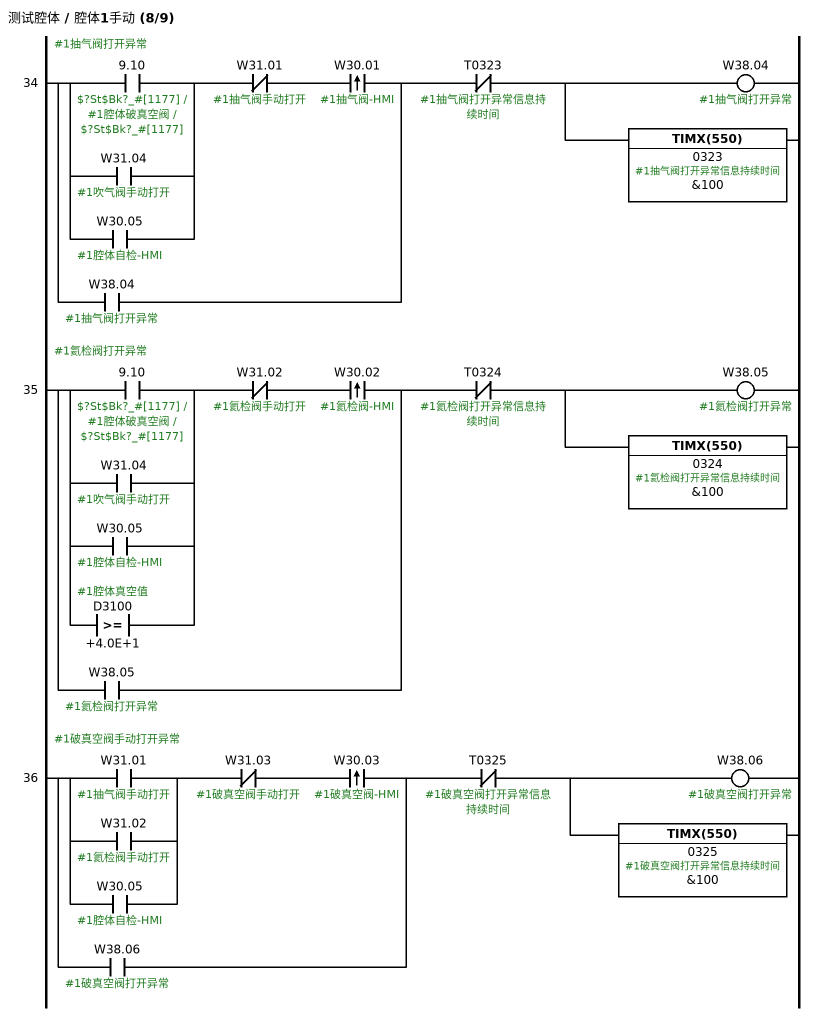
; [picture p120: 测试腔体 / 腔体1手动, rungs 34-36]
; rung 34: #1抽气阀打开异常
LD 9.10  ; $?St$Bk?_#[1177] / #1腔体破真空阀 / $?St$Bk?_#[1177]
OR W31.04  ; #1吹气阀手动打开
OR W30.05  ; #1腔体自检-HMI
ANDNOT W31.01  ; #1抽气阀手动打开
@AND W30.01  ; #1抽气阀-HMI
OR W38.04  ; #1抽气阀打开异常
ANDNOT T0323  ; #1抽气阀打开异常信息持续时间
OUT W38.04  ; #1抽气阀打开异常
TIMX(550) 0323 &100  ; #1抽气阀打开异常信息持续时间
; rung 35: #1氦检阀打开异常
LD 9.10  ; $?St$Bk?_#[1177] / #1腔体破真空阀 / $?St$Bk?_#[1177]
OR W31.04  ; #1吹气阀手动打开
OR W30.05  ; #1腔体自检-HMI
OR>=F(334) D3100 +4.0E+1  ; #1腔体真空值
ANDNOT W31.02  ; #1氦检阀手动打开
@AND W30.02  ; #1氦检阀-HMI
OR W38.05  ; #1氦检阀打开异常
ANDNOT T0324  ; #1氦检阀打开异常信息持续时间
OUT W38.05  ; #1氦检阀打开异常
TIMX(550) 0324 &100  ; #1氦检阀打开异常信息持续时间
; rung 36: #1破真空阀手动打开异常
LD W31.01  ; #1抽气阀手动打开
OR W31.02  ; #1氦检阀手动打开
OR W30.05  ; #1腔体自检-HMI
ANDNOT W31.03  ; #1破真空阀手动打开
@AND W30.03  ; #1破真空阀-HMI
OR W38.06  ; #1破真空阀打开异常
ANDNOT T0325  ; #1破真空阀打开异常信息持续时间
OUT W38.06  ; #1破真空阀打开异常
TIMX(550) 0325 &100  ; #1破真空阀打开异常信息持续时间

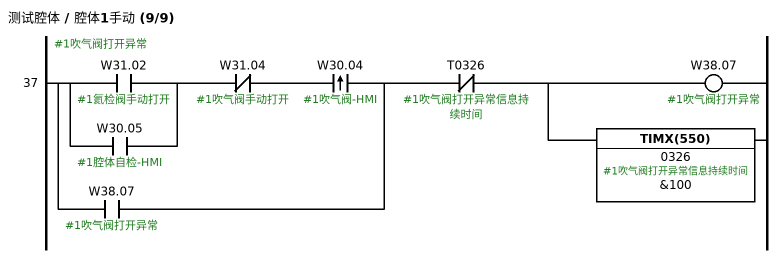
; rung 37: #1吹气阀打开异常
LD W31.02  ; #1氦检阀手动打开
OR W30.05  ; #1腔体自检-HMI
ANDNOT W31.04  ; #1吹气阀手动打开
@AND W30.04  ; #1吹气阀-HMI
OR W38.07  ; #1吹气阀打开异常
ANDNOT T0326  ; #1吹气阀打开异常信息持续时间
OUT W38.07  ; #1吹气阀打开异常
TIMX(550) 0326 &100  ; #1吹气阀打开异常信息持续时间

### Section 腔体2手动

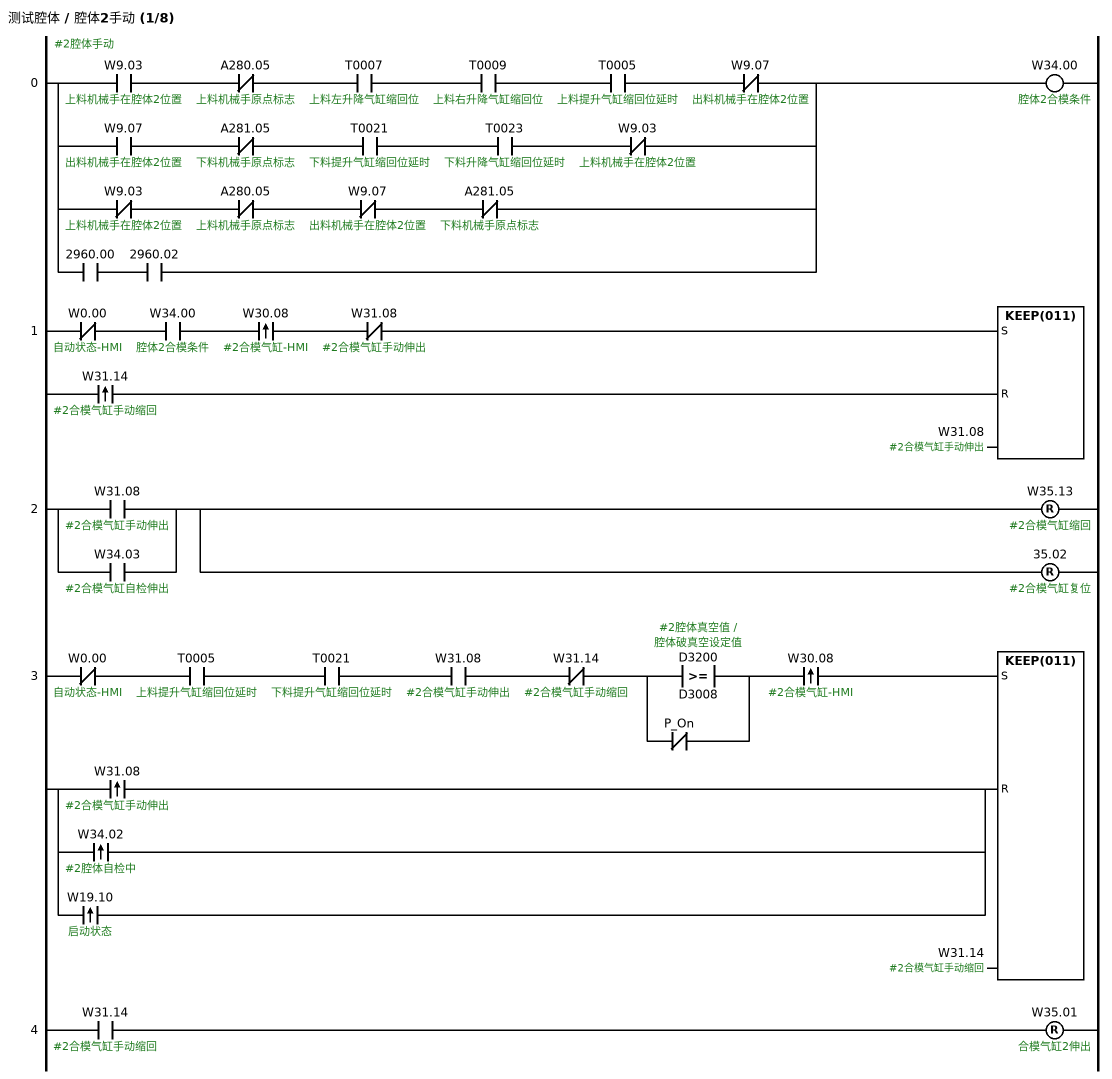
; rung 0: #2腔体手动
LD W9.03  ; 上料机械手在腔体2位置
ANDNOT A280.05  ; 上料机械手原点标志
AND T0007  ; 上料左升降气缸缩回位
AND T0009  ; 上料右升降气缸缩回位
AND T0005  ; 上料提升气缸缩回位延时
ANDNOT W9.07  ; 出料机械手在腔体2位置
LD W9.07  ; 出料机械手在腔体2位置
ANDNOT A281.05  ; 下料机械手原点标志
AND T0021  ; 下料提升气缸缩回位延时
AND T0023  ; 下料升降气缸缩回位延时
ANDNOT W9.03  ; 上料机械手在腔体2位置
ORLD
LDNOT W9.03  ; 上料机械手在腔体2位置
ANDNOT A280.05  ; 上料机械手原点标志
ANDNOT W9.07  ; 出料机械手在腔体2位置
ANDNOT A281.05  ; 下料机械手原点标志
ORLD
LD 2960.00
AND 2960.02
ORLD
OUT W34.00  ; 腔体2合模条件
; rung 1
LDNOT W0.00  ; 自动状态-HMI
AND W34.00  ; 腔体2合模条件
@AND W30.08  ; #2合模气缸-HMI
ANDNOT W31.08  ; #2合模气缸手动伸出
@LD W31.14  ; #2合模气缸手动缩回
KEEP(011) W31.08  ; #2合模气缸手动伸出
; rung 2
LD W31.08  ; #2合模气缸手动伸出
OR W34.03  ; #2合模气缸自检伸出
RSET W35.13  ; #2合模气缸缩回
RSET 35.02  ; #2合模气缸复位
; rung 3
LDNOT W0.00  ; 自动状态-HMI
AND T0005  ; 上料提升气缸缩回位延时
AND T0021  ; 下料提升气缸缩回位延时
AND W31.08  ; #2合模气缸手动伸出
ANDNOT W31.14  ; #2合模气缸手动缩回
LD>=F(334) D3200 D3008  ; #2腔体真空值, 腔体破真空设定值
ORNOT P_On
ANDLD
@AND W30.08  ; #2合模气缸-HMI
@LD W31.08  ; #2合模气缸手动伸出
@OR W34.02  ; #2腔体自检中
@OR W19.10  ; 启动状态
KEEP(011) W31.14  ; #2合模气缸手动缩回
; rung 4
LD W31.14  ; #2合模气缸手动缩回
RSET W35.01  ; 合模气缸2伸出

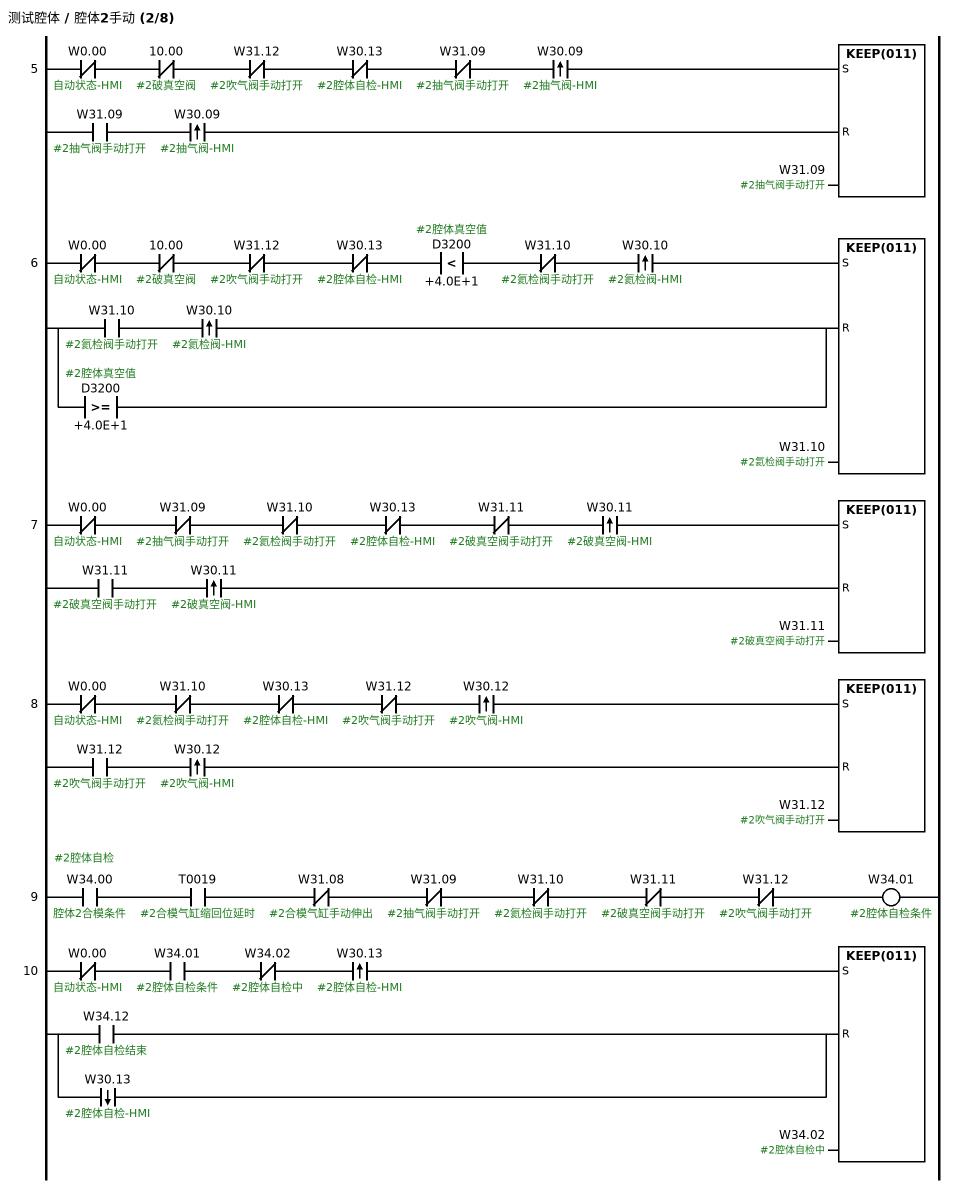
; rung 5
LDNOT W0.00  ; 自动状态-HMI
ANDNOT 10.00  ; #2破真空阀
ANDNOT W31.12  ; #2吹气阀手动打开
ANDNOT W30.13  ; #2腔体自检-HMI
ANDNOT W31.09  ; #2抽气阀手动打开
@AND W30.09  ; #2抽气阀-HMI
LD W31.09  ; #2抽气阀手动打开
@AND W30.09  ; #2抽气阀-HMI
KEEP(011) W31.09  ; #2抽气阀手动打开
; rung 6
LDNOT W0.00  ; 自动状态-HMI
ANDNOT 10.00  ; #2破真空阀
ANDNOT W31.12  ; #2吹气阀手动打开
ANDNOT W30.13  ; #2腔体自检-HMI
AND<F(331) D3200 +4.0E+1  ; #2腔体真空值
ANDNOT W31.10  ; #2氦检阀手动打开
@AND W30.10  ; #2氦检阀-HMI
LD W31.10  ; #2氦检阀手动打开
@AND W30.10  ; #2氦检阀-HMI
OR>=F(334) D3200 +4.0E+1  ; #2腔体真空值
KEEP(011) W31.10  ; #2氦检阀手动打开
; rung 7
LDNOT W0.00  ; 自动状态-HMI
ANDNOT W31.09  ; #2抽气阀手动打开
ANDNOT W31.10  ; #2氦检阀手动打开
ANDNOT W30.13  ; #2腔体自检-HMI
ANDNOT W31.11  ; #2破真空阀手动打开
@AND W30.11  ; #2破真空阀-HMI
LD W31.11  ; #2破真空阀手动打开
@AND W30.11  ; #2破真空阀-HMI
KEEP(011) W31.11  ; #2破真空阀手动打开
; rung 8
LDNOT W0.00  ; 自动状态-HMI
ANDNOT W31.10  ; #2氦检阀手动打开
ANDNOT W30.13  ; #2腔体自检-HMI
ANDNOT W31.12  ; #2吹气阀手动打开
@AND W30.12  ; #2吹气阀-HMI
LD W31.12  ; #2吹气阀手动打开
@AND W30.12  ; #2吹气阀-HMI
KEEP(011) W31.12  ; #2吹气阀手动打开
; rung 9: #2腔体自检
LD W34.00  ; 腔体2合模条件
AND T0019  ; #2合模气缸缩回位延时
ANDNOT W31.08  ; #2合模气缸手动伸出
ANDNOT W31.09  ; #2抽气阀手动打开
ANDNOT W31.10  ; #2氦检阀手动打开
ANDNOT W31.11  ; #2破真空阀手动打开
ANDNOT W31.12  ; #2吹气阀手动打开
OUT W34.01  ; #2腔体自检条件
; rung 10
LDNOT W0.00  ; 自动状态-HMI
AND W34.01  ; #2腔体自检条件
ANDNOT W34.02  ; #2腔体自检中
@AND W30.13  ; #2腔体自检-HMI
LD W34.12  ; #2腔体自检结束
%OR W30.13  ; #2腔体自检-HMI
KEEP(011) W34.02  ; #2腔体自检中

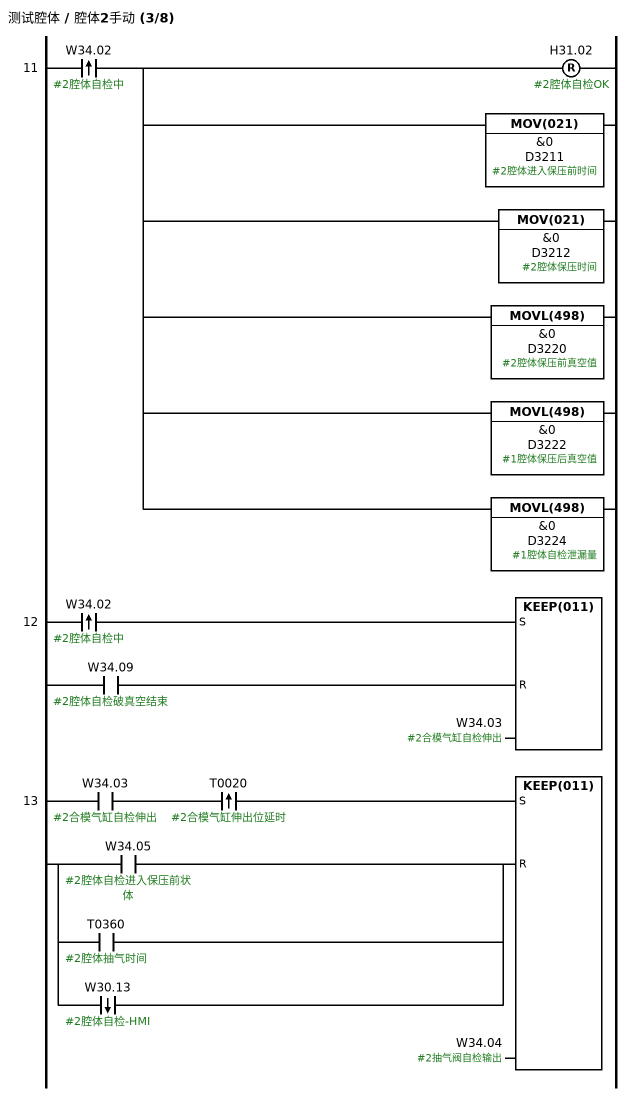
; rung 11
@LD W34.02  ; #2腔体自检中
RSET H31.02  ; #2腔体自检OK
MOV(021) &0 D3211  ; #2腔体进入保压前时间
MOV(021) &0 D3212  ; #2腔体保压时间
MOVL(498) &0 D3220  ; #2腔体保压前真空值
MOVL(498) &0 D3222  ; #1腔体保压后真空值
MOVL(498) &0 D3224  ; #1腔体自检泄漏量
; rung 12
@LD W34.02  ; #2腔体自检中
LD W34.09  ; #2腔体自检破真空结束
KEEP(011) W34.03  ; #2合模气缸自检伸出
; rung 13
LD W34.03  ; #2合模气缸自检伸出
@AND T0020  ; #2合模气缸伸出位延时
LD W34.05  ; #2腔体自检进入保压前状体
OR T0360  ; #2腔体抽气时间
%OR W30.13  ; #2腔体自检-HMI
KEEP(011) W34.04  ; #2抽气阀自检输出

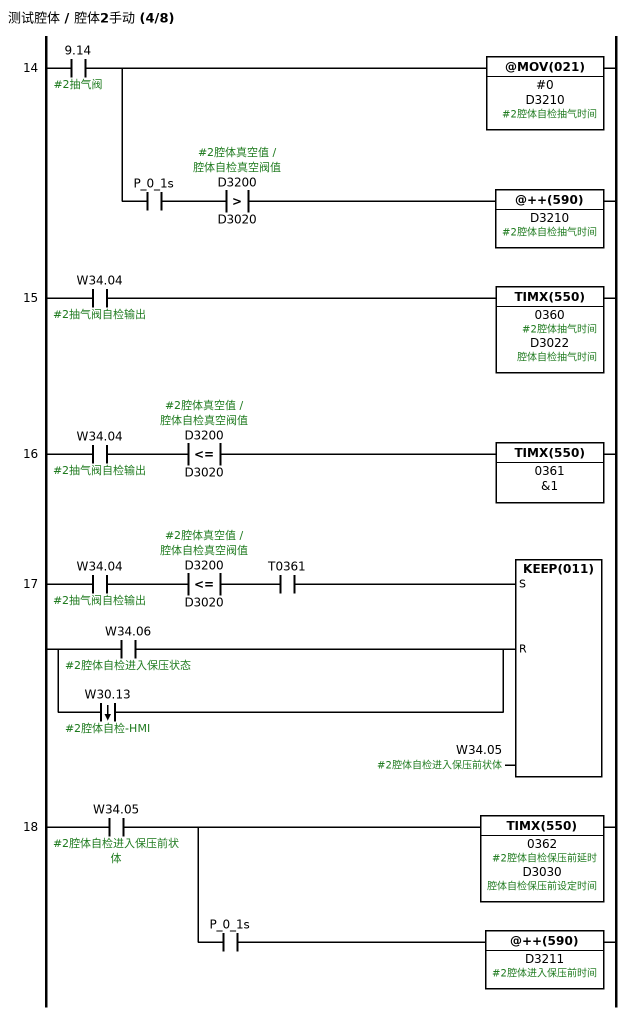
; rung 14
LD 9.14  ; #2抽气阀
@MOV(021) #0 D3210  ; #2腔体自检抽气时间
AND P_0_1s
AND>F(333) D3200 D3020  ; #2腔体真空值, 腔体自检真空阀值
@++(590) D3210  ; #2腔体自检抽气时间
; rung 15
LD W34.04  ; #2抽气阀自检输出
TIMX(550) 0360 D3022  ; 腔体自检抽气时间, #2腔体抽气时间
; rung 16
LD W34.04  ; #2抽气阀自检输出
AND<=F(332) D3200 D3020  ; #2腔体真空值, 腔体自检真空阀值
TIMX(550) 0361 &1
; rung 17
LD W34.04  ; #2抽气阀自检输出
AND<=F(332) D3200 D3020  ; #2腔体真空值, 腔体自检真空阀值
AND T0361
LD W34.06  ; #2腔体自检进入保压状态
%OR W30.13  ; #2腔体自检-HMI
KEEP(011) W34.05  ; #2腔体自检进入保压前状体
; rung 18
LD W34.05  ; #2腔体自检进入保压前状体
TIMX(550) 0362 D3030  ; 腔体自检保压前设定时间, #2腔体自检保压前延时
AND P_0_1s
@++(590) D3211  ; #2腔体进入保压前时间

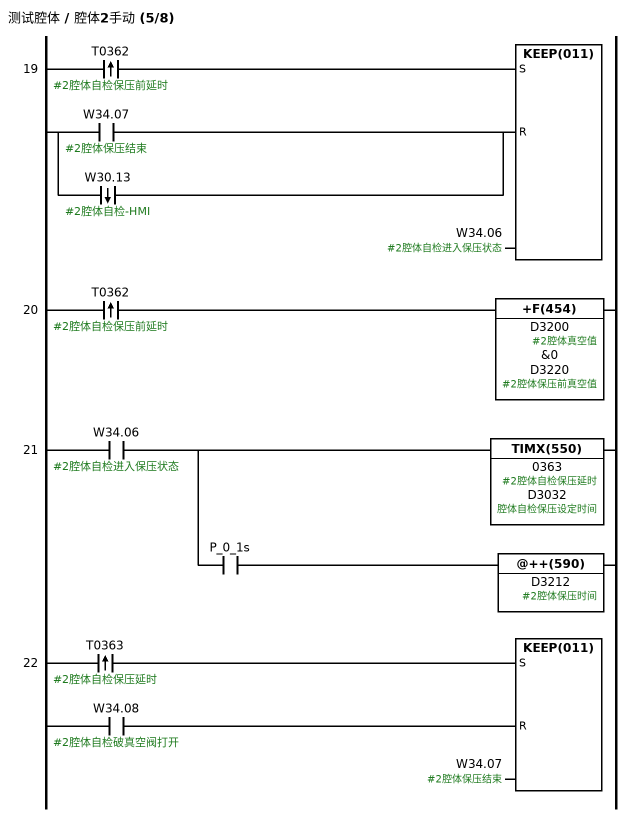
; rung 19
@LD T0362  ; #2腔体自检保压前延时
LD W34.07  ; #2腔体保压结束
%OR W30.13  ; #2腔体自检-HMI
KEEP(011) W34.06  ; #2腔体自检进入保压状态
; rung 20
@LD T0362  ; #2腔体自检保压前延时
+F(454) D3200 &0 D3220  ; #2腔体真空值, #2腔体保压前真空值
; rung 21
LD W34.06  ; #2腔体自检进入保压状态
TIMX(550) 0363 D3032  ; 腔体自检保压设定时间, #2腔体自检保压延时
AND P_0_1s
@++(590) D3212  ; #2腔体保压时间
; rung 22
@LD T0363  ; #2腔体自检保压延时
LD W34.08  ; #2腔体自检破真空阀打开
KEEP(011) W34.07  ; #2腔体保压结束

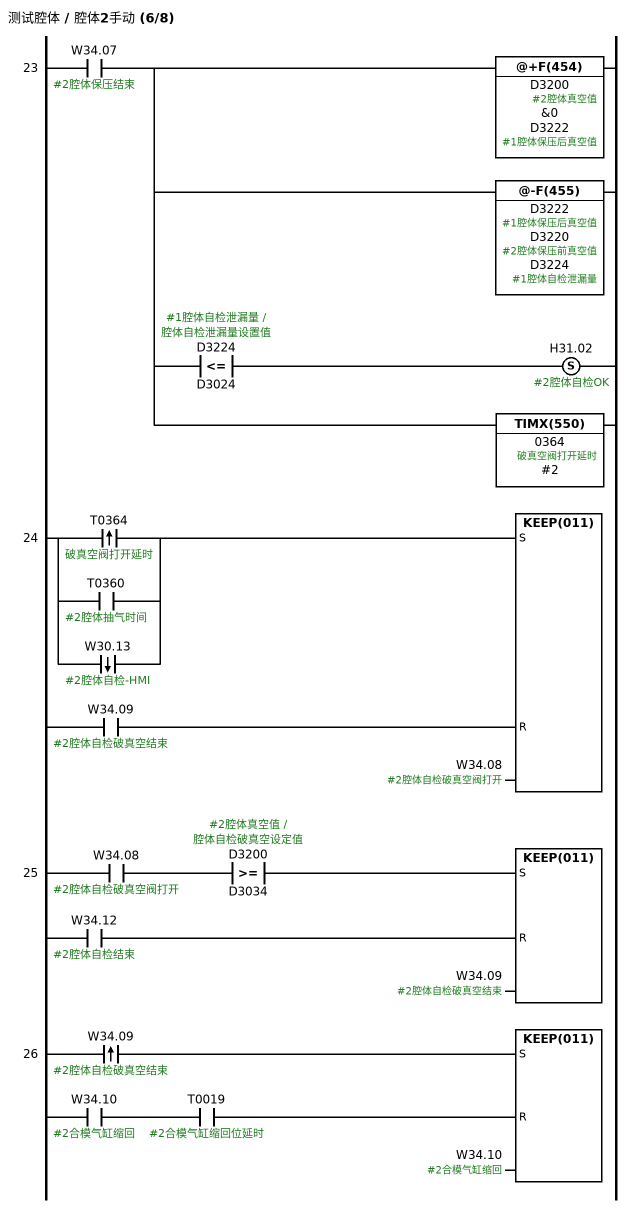
; rung 23
LD W34.07  ; #2腔体保压结束
OUT TR0
@+F(454) D3200 &0 D3222  ; #2腔体真空值, #1腔体保压后真空值
@-F(455) D3222 D3220 D3224  ; #1腔体保压后真空值, #2腔体保压前真空值, #1腔体自检泄漏量
AND<=(315) D3224 D3024  ; #1腔体自检泄漏量, 腔体自检泄漏量设置值
SET H31.02  ; #2腔体自检OK
LD TR0
TIMX(550) 0364 #2  ; 破真空阀打开延时
; rung 24
@LD T0364  ; 破真空阀打开延时
OR T0360  ; #2腔体抽气时间
%OR W30.13  ; #2腔体自检-HMI
LD W34.09  ; #2腔体自检破真空结束
KEEP(011) W34.08  ; #2腔体自检破真空阀打开
; rung 25
LD W34.08  ; #2腔体自检破真空阀打开
AND>=F(334) D3200 D3034  ; #2腔体真空值, 腔体自检破真空设定值
LD W34.12  ; #2腔体自检结束
KEEP(011) W34.09  ; #2腔体自检破真空结束
; rung 26
@LD W34.09  ; #2腔体自检破真空结束
LD W34.10  ; #2合模气缸缩回
AND T0019  ; #2合模气缸缩回位延时
KEEP(011) W34.10  ; #2合模气缸缩回

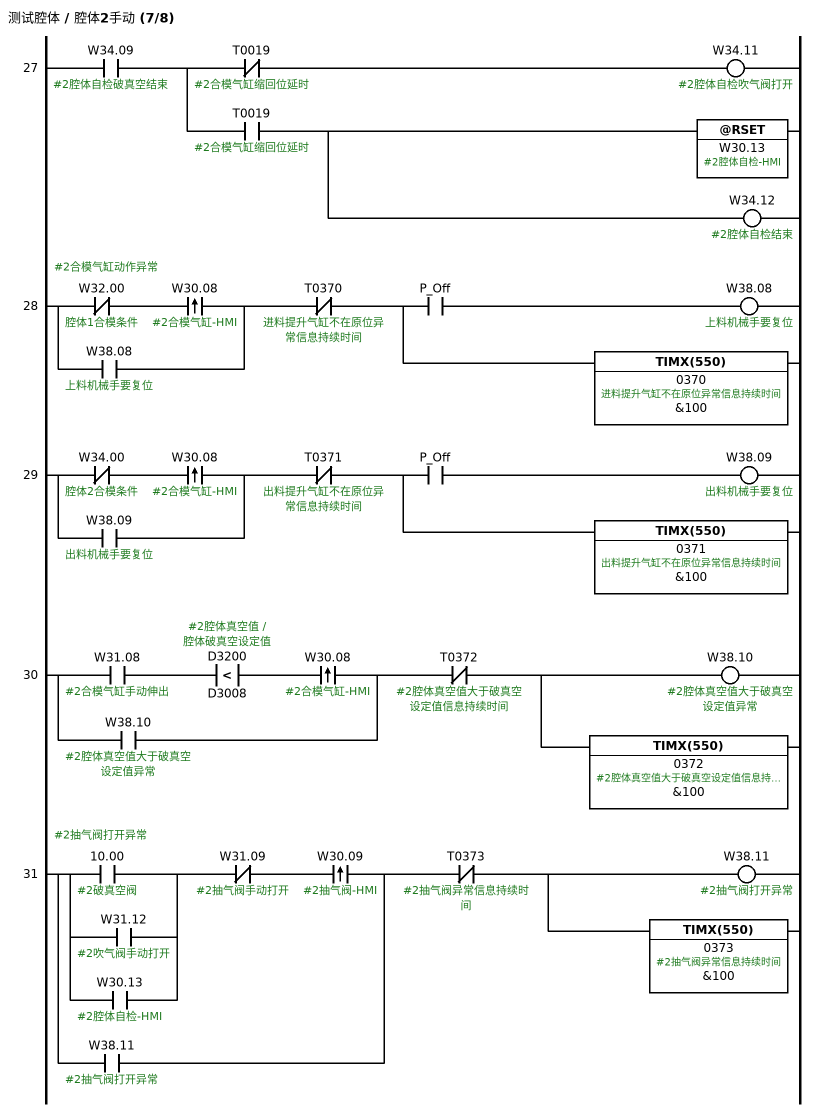
; rung 27
LD W34.09  ; #2腔体自检破真空结束
OUT TR0
ANDNOT T0019  ; #2合模气缸缩回位延时
OUT W34.11  ; #2腔体自检吹气阀打开
LD TR0
AND T0019  ; #2合模气缸缩回位延时
@RSET W30.13  ; #2腔体自检-HMI
OUT W34.12  ; #2腔体自检结束
; rung 28: #2合模气缸动作异常
LDNOT W32.00  ; 腔体1合模条件
@AND W30.08  ; #2合模气缸-HMI
OR W38.08  ; 上料机械手要复位
ANDNOT T0370  ; 进料提升气缸不在原位异常信息持续时间
OUT TR0
AND P_Off
OUT W38.08  ; 上料机械手要复位
LD TR0
TIMX(550) 0370 &100  ; 进料提升气缸不在原位异常信息持续时间
; rung 29
LDNOT W34.00  ; 腔体2合模条件
@AND W30.08  ; #2合模气缸-HMI
OR W38.09  ; 出料机械手要复位
ANDNOT T0371  ; 出料提升气缸不在原位异常信息持续时间
OUT TR0
AND P_Off
OUT W38.09  ; 出料机械手要复位
LD TR0
TIMX(550) 0371 &100  ; 出料提升气缸不在原位异常信息持续时间
; rung 30
LD W31.08  ; #2合模气缸手动伸出
AND<F(331) D3200 D3008  ; #2腔体真空值, 腔体破真空设定值
@AND W30.08  ; #2合模气缸-HMI
OR W38.10  ; #2腔体真空值大于破真空设定值异常
ANDNOT T0372  ; #2腔体真空值大于破真空设定值信息持续时间
OUT W38.10  ; #2腔体真空值大于破真空设定值异常
TIMX(550) 0372 &100  ; #2腔体真空值大于破真空设定值信息持续时间
; rung 31: #2抽气阀打开异常
LD 10.00  ; #2破真空阀
OR W31.12  ; #2吹气阀手动打开
OR W30.13  ; #2腔体自检-HMI
ANDNOT W31.09  ; #2抽气阀手动打开
@AND W30.09  ; #2抽气阀-HMI
OR W38.11  ; #2抽气阀打开异常
ANDNOT T0373  ; #2抽气阀异常信息持续时间
OUT W38.11  ; #2抽气阀打开异常
TIMX(550) 0373 &100  ; #2抽气阀异常信息持续时间

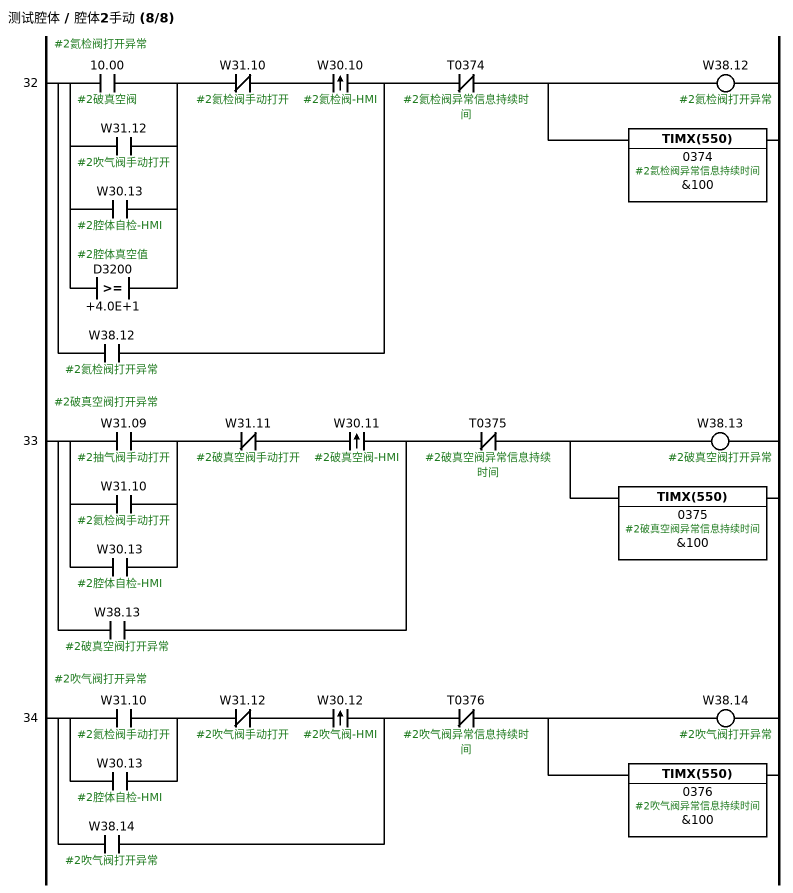
; rung 32: #2氦检阀打开异常
LD 10.00  ; #2破真空阀
OR W31.12  ; #2吹气阀手动打开
OR W30.13  ; #2腔体自检-HMI
OR>=F(334) D3200 +4.0E+1  ; #2腔体真空值
ANDNOT W31.10  ; #2氦检阀手动打开
@AND W30.10  ; #2氦检阀-HMI
OR W38.12  ; #2氦检阀打开异常
ANDNOT T0374  ; #2氦检阀异常信息持续时间
OUT W38.12  ; #2氦检阀打开异常
TIMX(550) 0374 &100  ; #2氦检阀异常信息持续时间
; rung 33: #2破真空阀打开异常
LD W31.09  ; #2抽气阀手动打开
OR W31.10  ; #2氦检阀手动打开
OR W30.13  ; #2腔体自检-HMI
ANDNOT W31.11  ; #2破真空阀手动打开
@AND W30.11  ; #2破真空阀-HMI
OR W38.13  ; #2破真空阀打开异常
ANDNOT T0375  ; #2破真空阀异常信息持续时间
OUT W38.13  ; #2破真空阀打开异常
TIMX(550) 0375 &100  ; #2破真空阀异常信息持续时间
; rung 34: #2吹气阀打开异常
LD W31.10  ; #2氦检阀手动打开
OR W30.13  ; #2腔体自检-HMI
ANDNOT W31.12  ; #2吹气阀手动打开
@AND W30.12  ; #2吹气阀-HMI
OR W38.14  ; #2吹气阀打开异常
ANDNOT T0376  ; #2吹气阀异常信息持续时间
OUT W38.14  ; #2吹气阀打开异常
TIMX(550) 0376 &100  ; #2吹气阀异常信息持续时间

### Section 腔体1自动

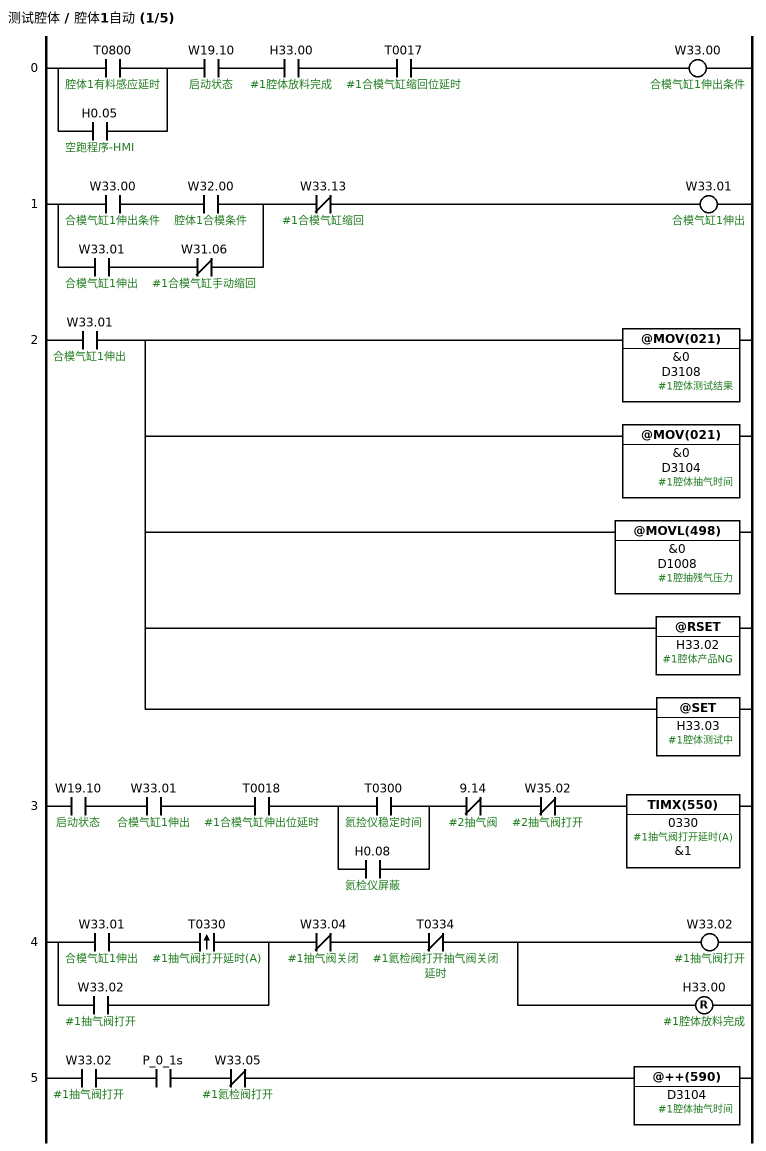
; rung 0
LD T0800  ; 腔体1有料感应延时
OR H0.05  ; 空跑程序-HMI
AND W19.10  ; 启动状态
AND H33.00  ; #1腔体放料完成
AND T0017  ; #1合模气缸缩回位延时
OUT W33.00  ; 合模气缸1伸出条件
; rung 1
LD W33.00  ; 合模气缸1伸出条件
AND W32.00  ; 腔体1合模条件
LD W33.01  ; 合模气缸1伸出
ANDNOT W31.06  ; #1合模气缸手动缩回
ORLD
ANDNOT W33.13  ; #1合模气缸缩回
OUT W33.01  ; 合模气缸1伸出
; rung 2
LD W33.01  ; 合模气缸1伸出
@MOV(021) &0 D3108  ; #1腔体测试结果
@MOV(021) &0 D3104  ; #1腔体抽气时间
@MOVL(498) &0 D1008  ; #1腔抽残气压力
@RSET H33.02  ; #1腔体产品NG
@SET H33.03  ; #1腔体测试中
; rung 3
LD W19.10  ; 启动状态
AND W33.01  ; 合模气缸1伸出
AND T0018  ; #1合模气缸伸出位延时
LD T0300  ; 氦捡仪稳定时间
OR H0.08  ; 氦检仪屏蔽
ANDLD
ANDNOT 9.14  ; #2抽气阀
ANDNOT W35.02  ; #2抽气阀打开
TIMX(550) 0330 &1  ; #1抽气阀打开延时(A)
; rung 4
LD W33.01  ; 合模气缸1伸出
@AND T0330  ; #1抽气阀打开延时(A)
OR W33.02  ; #1抽气阀打开
ANDNOT W33.04  ; #1抽气阀关闭
ANDNOT T0334  ; #1氦检阀打开抽气阀关闭延时
OUT W33.02  ; #1抽气阀打开
RSET H33.00  ; #1腔体放料完成
; rung 5
LD W33.02  ; #1抽气阀打开
AND P_0_1s
ANDNOT W33.05  ; #1氦检阀打开
@++(590) D3104  ; #1腔体抽气时间

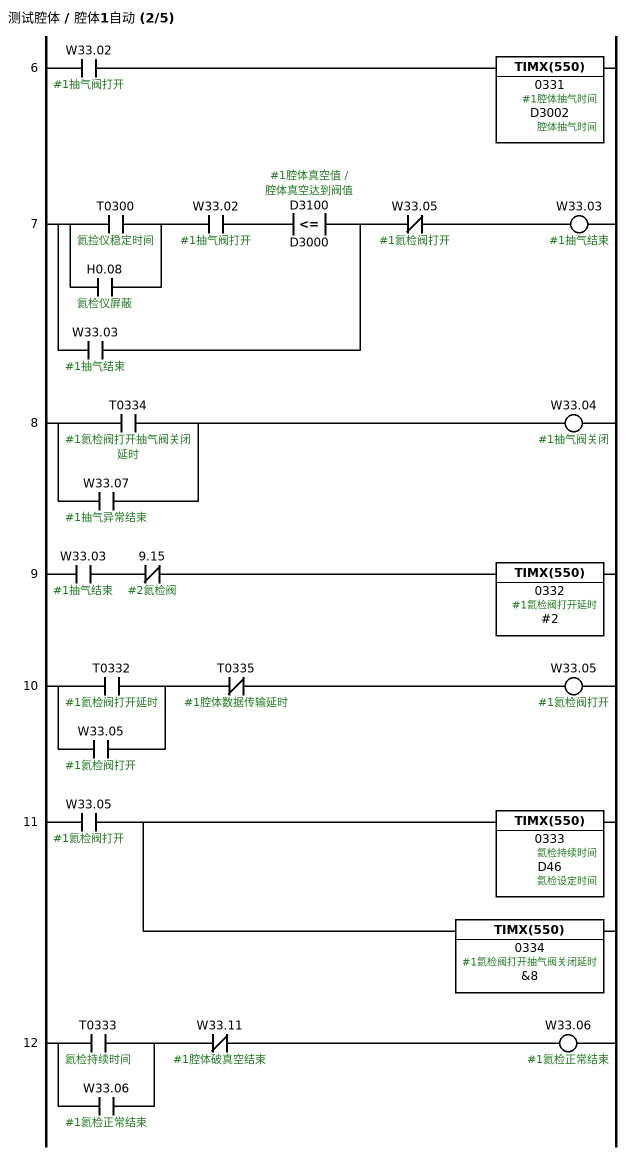
; rung 6
LD W33.02  ; #1抽气阀打开
TIMX(550) 0331 D3002  ; 腔体抽气时间, #1腔体抽气时间
; rung 7
LD T0300  ; 氦捡仪稳定时间
OR H0.08  ; 氦检仪屏蔽
AND W33.02  ; #1抽气阀打开
AND<=F(332) D3100 D3000  ; #1腔体真空值, 腔体真空达到阀值
OR W33.03  ; #1抽气结束
ANDNOT W33.05  ; #1氦检阀打开
OUT W33.03  ; #1抽气结束
; rung 8
LD T0334  ; #1氦检阀打开抽气阀关闭延时
OR W33.07  ; #1抽气异常结束
OUT W33.04  ; #1抽气阀关闭
; rung 9
LD W33.03  ; #1抽气结束
ANDNOT 9.15  ; #2氦检阀
TIMX(550) 0332 #2  ; #1氦检阀打开延时
; rung 10
LD T0332  ; #1氦检阀打开延时
OR W33.05  ; #1氦检阀打开
ANDNOT T0335  ; #1腔体数据传输延时
OUT W33.05  ; #1氦检阀打开
; rung 11
LD W33.05  ; #1氦检阀打开
TIMX(550) 0333 D46  ; 氦检设定时间, 氦检持续时间
TIMX(550) 0334 &8  ; #1氦检阀打开抽气阀关闭延时
; rung 12
LD T0333  ; 氦检持续时间
OR W33.06  ; #1氦检正常结束
ANDNOT W33.11  ; #1腔体破真空结束
OUT W33.06  ; #1氦检正常结束

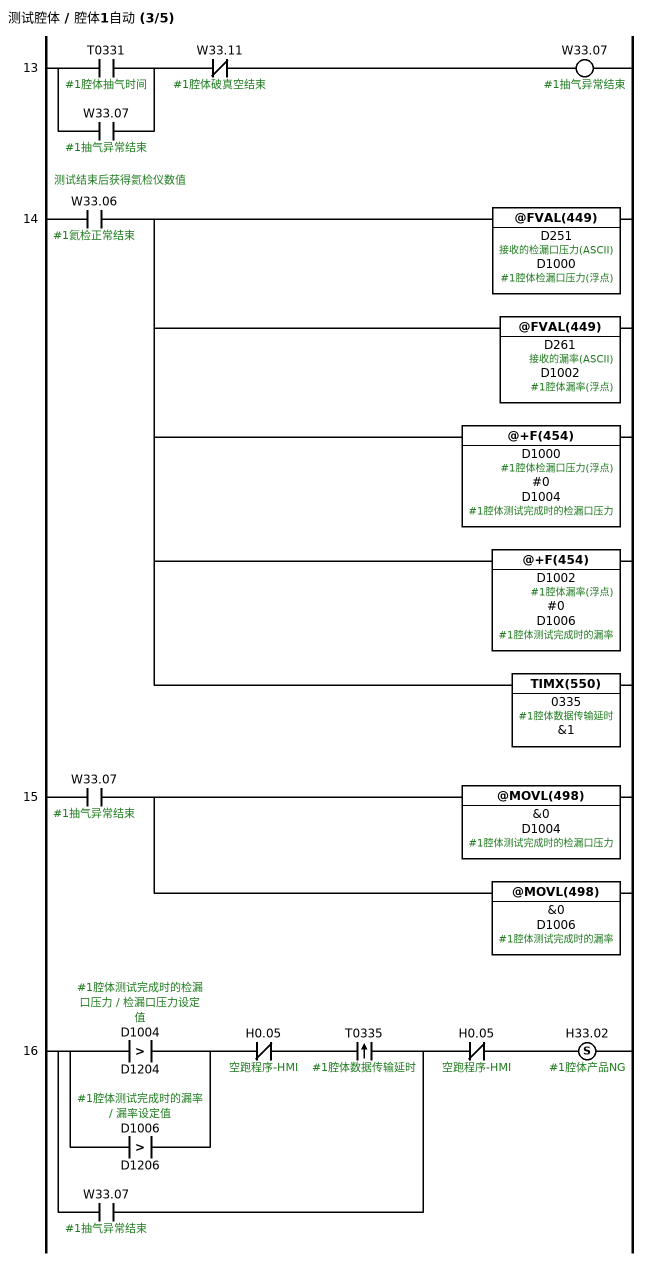
; rung 13
LD T0331  ; #1腔体抽气时间
OR W33.07  ; #1抽气异常结束
ANDNOT W33.11  ; #1腔体破真空结束
OUT W33.07  ; #1抽气异常结束
; rung 14: 测试结束后获得氦检仪数值
LD W33.06  ; #1氦检正常结束
@FVAL(449) D251 D1000  ; 接收的检漏口压力(ASCII), #1腔体检漏口压力(浮点)
@FVAL(449) D261 D1002  ; 接收的漏率(ASCII), #1腔体漏率(浮点)
@+F(454) D1000 #0 D1004  ; #1腔体检漏口压力(浮点), #1腔体测试完成时的检漏口压力
@+F(454) D1002 #0 D1006  ; #1腔体漏率(浮点), #1腔体测试完成时的漏率
TIMX(550) 0335 &1  ; #1腔体数据传输延时
; rung 15
LD W33.07  ; #1抽气异常结束
@MOVL(498) &0 D1004  ; #1腔体测试完成时的检漏口压力
@MOVL(498) &0 D1006  ; #1腔体测试完成时的漏率
; rung 16
LD>F(333) D1004 D1204  ; #1腔体测试完成时的检漏口压力, 检漏口压力设定值
OR>F(333) D1006 D1206  ; #1腔体测试完成时的漏率, 漏率设定值
ANDNOT H0.05  ; 空跑程序-HMI
@AND T0335  ; #1腔体数据传输延时
OR W33.07  ; #1抽气异常结束
ANDNOT H0.05  ; 空跑程序-HMI
SET H33.02  ; #1腔体产品NG

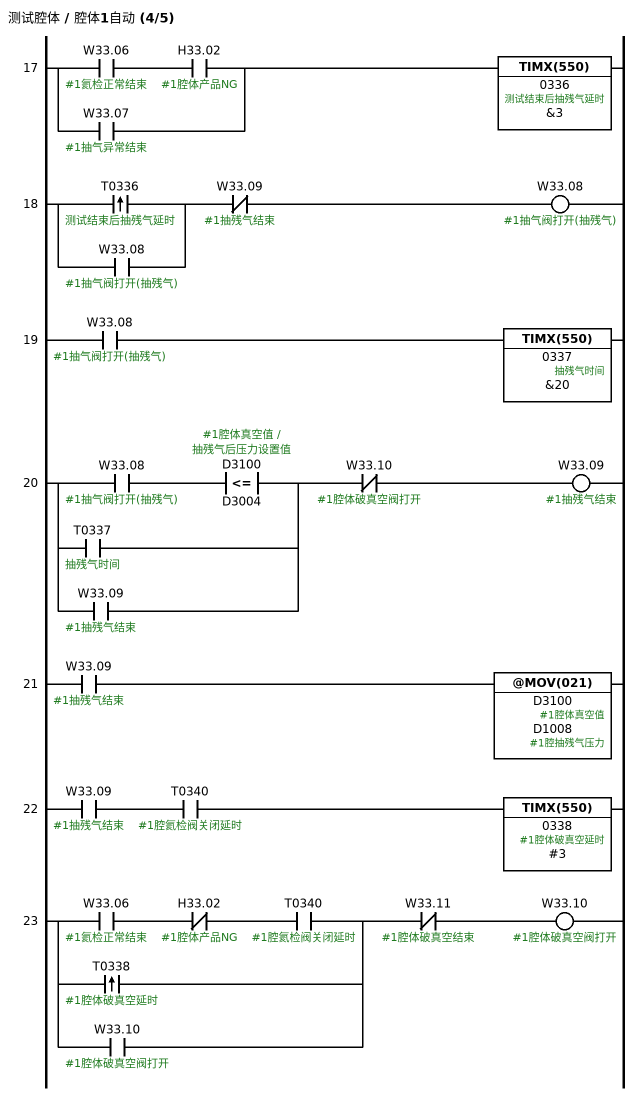
; rung 17
LD W33.06  ; #1氦检正常结束
AND H33.02  ; #1腔体产品NG
OR W33.07  ; #1抽气异常结束
TIMX(550) 0336 &3  ; 测试结束后抽残气延时
; rung 18
@LD T0336  ; 测试结束后抽残气延时
OR W33.08  ; #1抽气阀打开(抽残气)
ANDNOT W33.09  ; #1抽残气结束
OUT W33.08  ; #1抽气阀打开(抽残气)
; rung 19
LD W33.08  ; #1抽气阀打开(抽残气)
TIMX(550) 0337 &20  ; 抽残气时间
; rung 20
LD W33.08  ; #1抽气阀打开(抽残气)
AND<=F(332) D3100 D3004  ; #1腔体真空值, 抽残气后压力设置值
OR T0337  ; 抽残气时间
OR W33.09  ; #1抽残气结束
ANDNOT W33.10  ; #1腔体破真空阀打开
OUT W33.09  ; #1抽残气结束
; rung 21
LD W33.09  ; #1抽残气结束
@MOV(021) D3100 D1008  ; #1腔体真空值, #1腔抽残气压力
; rung 22
LD W33.09  ; #1抽残气结束
AND T0340  ; #1腔氦检阀关闭延时
TIMX(550) 0338 #3  ; #1腔体破真空延时
; rung 23
LD W33.06  ; #1氦检正常结束
ANDNOT H33.02  ; #1腔体产品NG
AND T0340  ; #1腔氦检阀关闭延时
@OR T0338  ; #1腔体破真空延时
OR W33.10  ; #1腔体破真空阀打开
ANDNOT W33.11  ; #1腔体破真空结束
OUT W33.10  ; #1腔体破真空阀打开

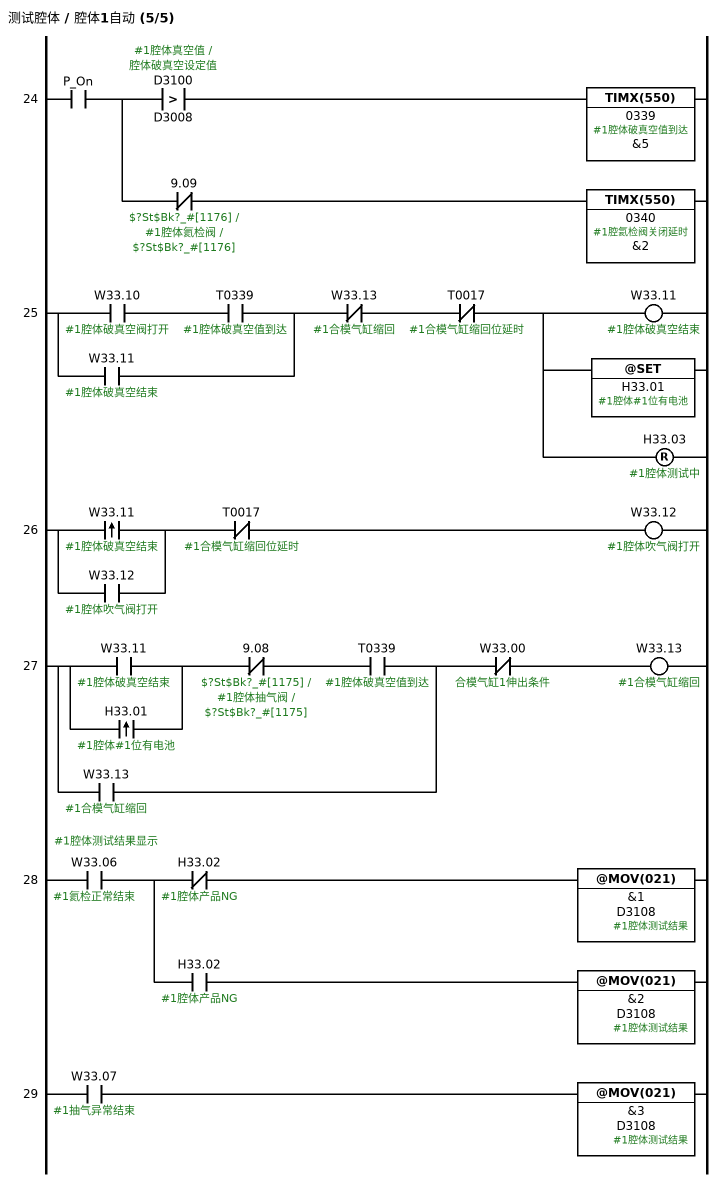
; rung 24
LD P_On
OUT TR0
AND>F(333) D3100 D3008  ; #1腔体真空值, 腔体破真空设定值
TIMX(550) 0339 &5  ; #1腔体破真空值到达
LD TR0
ANDNOT 9.09  ; $?St$Bk?_#[1176] / #1腔体氦检阀 / $?St$Bk?_#[1176]
TIMX(550) 0340 &2  ; #1腔氦检阀关闭延时
; rung 25
LD W33.10  ; #1腔体破真空阀打开
AND T0339  ; #1腔体破真空值到达
OR W33.11  ; #1腔体破真空结束
ANDNOT W33.13  ; #1合模气缸缩回
ANDNOT T0017  ; #1合模气缸缩回位延时
OUT W33.11  ; #1腔体破真空结束
@SET H33.01  ; #1腔体#1位有电池
RSET H33.03  ; #1腔体测试中
; rung 26
@LD W33.11  ; #1腔体破真空结束
OR W33.12  ; #1腔体吹气阀打开
ANDNOT T0017  ; #1合模气缸缩回位延时
OUT W33.12  ; #1腔体吹气阀打开
; rung 27
LD W33.11  ; #1腔体破真空结束
@OR H33.01  ; #1腔体#1位有电池
ANDNOT 9.08  ; $?St$Bk?_#[1175] / #1腔体抽气阀 / $?St$Bk?_#[1175]
AND T0339  ; #1腔体破真空值到达
OR W33.13  ; #1合模气缸缩回
ANDNOT W33.00  ; 合模气缸1伸出条件
OUT W33.13  ; #1合模气缸缩回
; rung 28: #1腔体测试结果显示
LD W33.06  ; #1氦检正常结束
OUT TR0
ANDNOT H33.02  ; #1腔体产品NG
@MOV(021) &1 D3108  ; #1腔体测试结果
LD TR0
AND H33.02  ; #1腔体产品NG
@MOV(021) &2 D3108  ; #1腔体测试结果
; rung 29
LD W33.07  ; #1抽气异常结束
@MOV(021) &3 D3108  ; #1腔体测试结果

### Section 腔体2自动

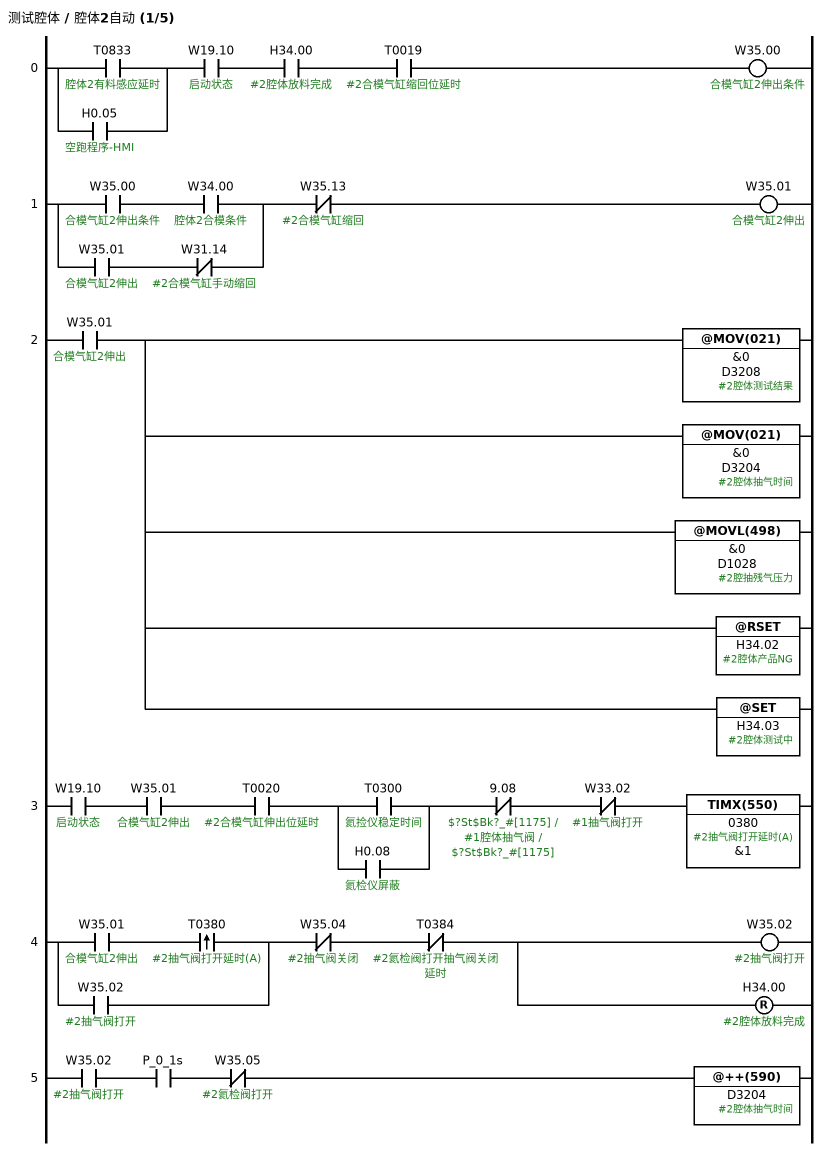
; rung 0
LD T0833  ; 腔体2有料感应延时
OR H0.05  ; 空跑程序-HMI
AND W19.10  ; 启动状态
AND H34.00  ; #2腔体放料完成
AND T0019  ; #2合模气缸缩回位延时
OUT W35.00  ; 合模气缸2伸出条件
; rung 1
LD W35.00  ; 合模气缸2伸出条件
AND W34.00  ; 腔体2合模条件
LD W35.01  ; 合模气缸2伸出
ANDNOT W31.14  ; #2合模气缸手动缩回
ORLD
ANDNOT W35.13  ; #2合模气缸缩回
OUT W35.01  ; 合模气缸2伸出
; rung 2
LD W35.01  ; 合模气缸2伸出
@MOV(021) &0 D3208  ; #2腔体测试结果
@MOV(021) &0 D3204  ; #2腔体抽气时间
@MOVL(498) &0 D1028  ; #2腔抽残气压力
@RSET H34.02  ; #2腔体产品NG
@SET H34.03  ; #2腔体测试中
; rung 3
LD W19.10  ; 启动状态
AND W35.01  ; 合模气缸2伸出
AND T0020  ; #2合模气缸伸出位延时
LD T0300  ; 氦捡仪稳定时间
OR H0.08  ; 氦检仪屏蔽
ANDLD
ANDNOT 9.08  ; $?St$Bk?_#[1175] / #1腔体抽气阀 / $?St$Bk?_#[1175]
ANDNOT W33.02  ; #1抽气阀打开
TIMX(550) 0380 &1  ; #2抽气阀打开延时(A)
; rung 4
LD W35.01  ; 合模气缸2伸出
@AND T0380  ; #2抽气阀打开延时(A)
OR W35.02  ; #2抽气阀打开
ANDNOT W35.04  ; #2抽气阀关闭
ANDNOT T0384  ; #2氦检阀打开抽气阀关闭延时
OUT W35.02  ; #2抽气阀打开
RSET H34.00  ; #2腔体放料完成
; rung 5
LD W35.02  ; #2抽气阀打开
AND P_0_1s
ANDNOT W35.05  ; #2氦检阀打开
@++(590) D3204  ; #2腔体抽气时间

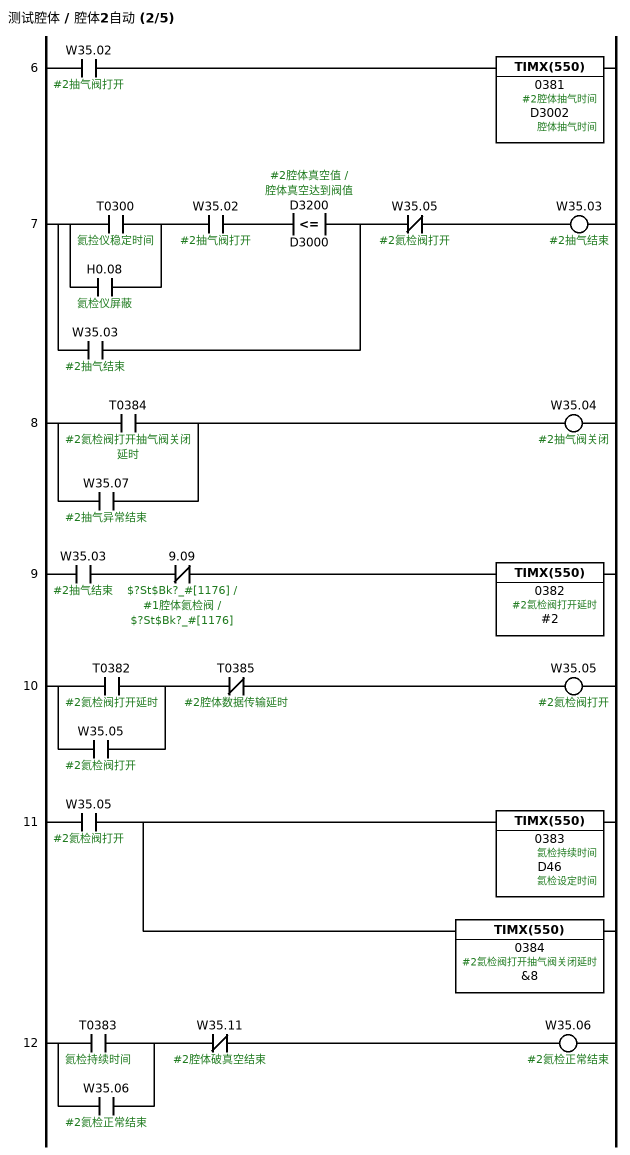
; rung 6
LD W35.02  ; #2抽气阀打开
TIMX(550) 0381 D3002  ; 腔体抽气时间, #2腔体抽气时间
; rung 7
LD T0300  ; 氦捡仪稳定时间
OR H0.08  ; 氦检仪屏蔽
AND W35.02  ; #2抽气阀打开
AND<=F(332) D3200 D3000  ; #2腔体真空值, 腔体真空达到阀值
OR W35.03  ; #2抽气结束
ANDNOT W35.05  ; #2氦检阀打开
OUT W35.03  ; #2抽气结束
; rung 8
LD T0384  ; #2氦检阀打开抽气阀关闭延时
OR W35.07  ; #2抽气异常结束
OUT W35.04  ; #2抽气阀关闭
; rung 9
LD W35.03  ; #2抽气结束
ANDNOT 9.09  ; $?St$Bk?_#[1176] / #1腔体氦检阀 / $?St$Bk?_#[1176]
TIMX(550) 0382 #2  ; #2氦检阀打开延时
; rung 10
LD T0382  ; #2氦检阀打开延时
OR W35.05  ; #2氦检阀打开
ANDNOT T0385  ; #2腔体数据传输延时
OUT W35.05  ; #2氦检阀打开
; rung 11
LD W35.05  ; #2氦检阀打开
TIMX(550) 0383 D46  ; 氦检设定时间, 氦检持续时间
TIMX(550) 0384 &8  ; #2氦检阀打开抽气阀关闭延时
; rung 12
LD T0383  ; 氦检持续时间
OR W35.06  ; #2氦检正常结束
ANDNOT W35.11  ; #2腔体破真空结束
OUT W35.06  ; #2氦检正常结束

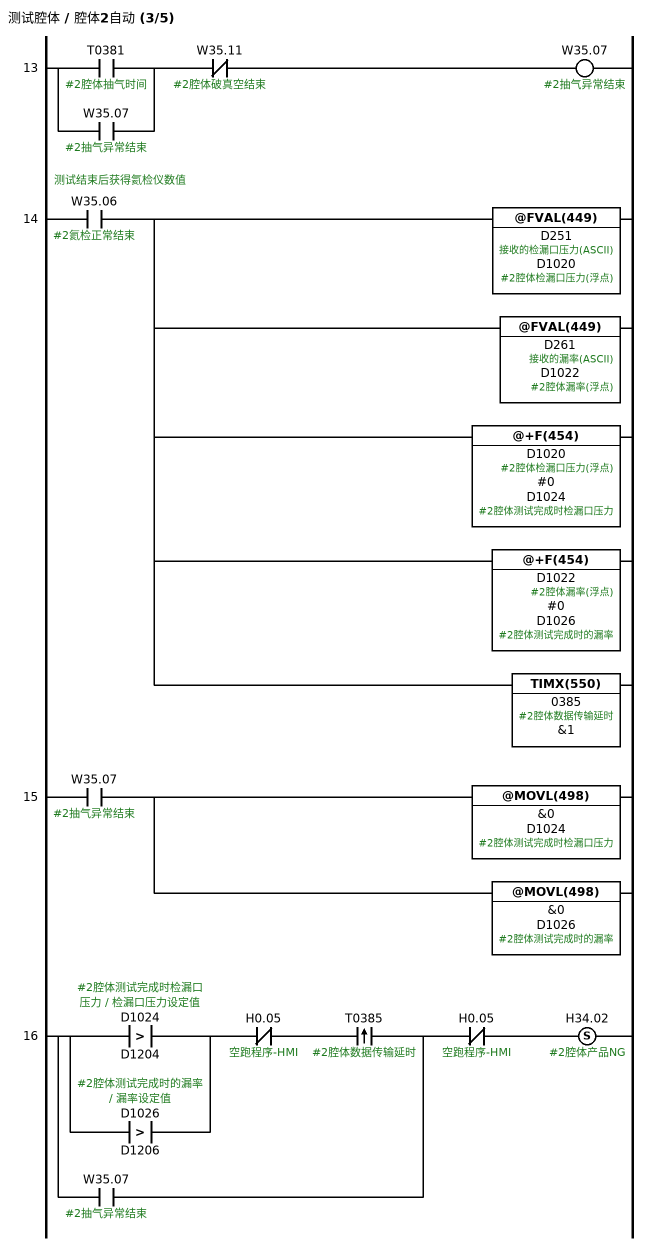
; rung 13
LD T0381  ; #2腔体抽气时间
OR W35.07  ; #2抽气异常结束
ANDNOT W35.11  ; #2腔体破真空结束
OUT W35.07  ; #2抽气异常结束
; rung 14: 测试结束后获得氦检仪数值
LD W35.06  ; #2氦检正常结束
@FVAL(449) D251 D1020  ; 接收的检漏口压力(ASCII), #2腔体检漏口压力(浮点)
@FVAL(449) D261 D1022  ; 接收的漏率(ASCII), #2腔体漏率(浮点)
@+F(454) D1020 #0 D1024  ; #2腔体检漏口压力(浮点), #2腔体测试完成时检漏口压力
@+F(454) D1022 #0 D1026  ; #2腔体漏率(浮点), #2腔体测试完成时的漏率
TIMX(550) 0385 &1  ; #2腔体数据传输延时
; rung 15
LD W35.07  ; #2抽气异常结束
@MOVL(498) &0 D1024  ; #2腔体测试完成时检漏口压力
@MOVL(498) &0 D1026  ; #2腔体测试完成时的漏率
; rung 16
LD>F(333) D1024 D1204  ; #2腔体测试完成时检漏口压力, 检漏口压力设定值
OR>F(333) D1026 D1206  ; #2腔体测试完成时的漏率, 漏率设定值
ANDNOT H0.05  ; 空跑程序-HMI
@AND T0385  ; #2腔体数据传输延时
OR W35.07  ; #2抽气异常结束
ANDNOT H0.05  ; 空跑程序-HMI
SET H34.02  ; #2腔体产品NG

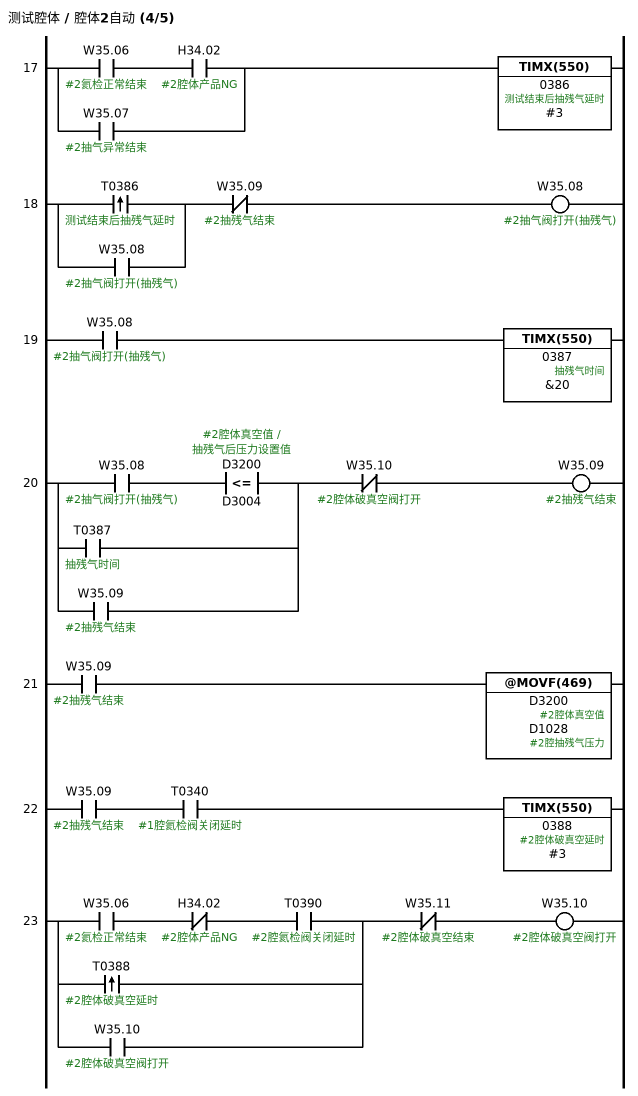
; rung 17
LD W35.06  ; #2氦检正常结束
AND H34.02  ; #2腔体产品NG
OR W35.07  ; #2抽气异常结束
TIMX(550) 0386 #3  ; 测试结束后抽残气延时
; rung 18
@LD T0386  ; 测试结束后抽残气延时
OR W35.08  ; #2抽气阀打开(抽残气)
ANDNOT W35.09  ; #2抽残气结束
OUT W35.08  ; #2抽气阀打开(抽残气)
; rung 19
LD W35.08  ; #2抽气阀打开(抽残气)
TIMX(550) 0387 &20  ; 抽残气时间
; rung 20
LD W35.08  ; #2抽气阀打开(抽残气)
AND<=F(332) D3200 D3004  ; #2腔体真空值, 抽残气后压力设置值
OR T0387  ; 抽残气时间
OR W35.09  ; #2抽残气结束
ANDNOT W35.10  ; #2腔体破真空阀打开
OUT W35.09  ; #2抽残气结束
; rung 21
LD W35.09  ; #2抽残气结束
@MOVF(469) D3200 D1028  ; #2腔体真空值, #2腔抽残气压力
; rung 22
LD W35.09  ; #2抽残气结束
AND T0340  ; #1腔氦检阀关闭延时
TIMX(550) 0388 #3  ; #2腔体破真空延时
; rung 23
LD W35.06  ; #2氦检正常结束
ANDNOT H34.02  ; #2腔体产品NG
AND T0390  ; #2腔氦检阀关闭延时
@OR T0388  ; #2腔体破真空延时
OR W35.10  ; #2腔体破真空阀打开
ANDNOT W35.11  ; #2腔体破真空结束
OUT W35.10  ; #2腔体破真空阀打开

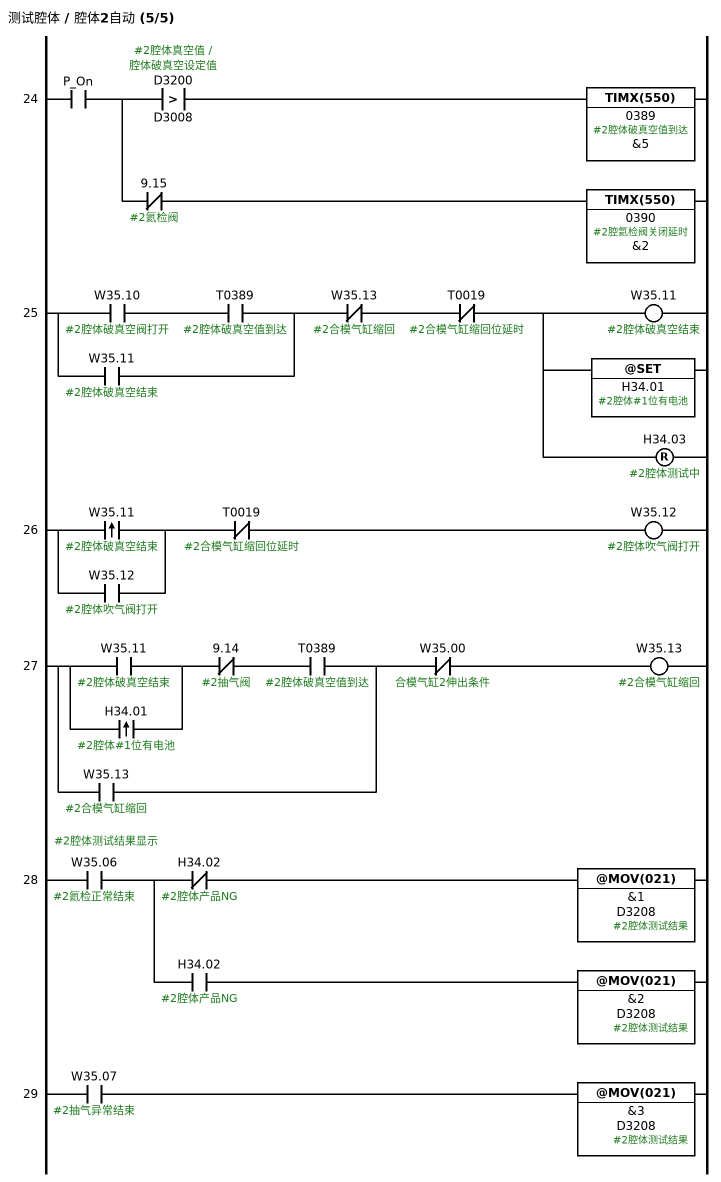
; rung 24
LD P_On
OUT TR0
AND>F(333) D3200 D3008  ; #2腔体真空值, 腔体破真空设定值
TIMX(550) 0389 &5  ; #2腔体破真空值到达
LD TR0
ANDNOT 9.15  ; #2氦检阀
TIMX(550) 0390 &2  ; #2腔氦检阀关闭延时
; rung 25
LD W35.10  ; #2腔体破真空阀打开
AND T0389  ; #2腔体破真空值到达
OR W35.11  ; #2腔体破真空结束
ANDNOT W35.13  ; #2合模气缸缩回
ANDNOT T0019  ; #2合模气缸缩回位延时
OUT W35.11  ; #2腔体破真空结束
@SET H34.01  ; #2腔体#1位有电池
RSET H34.03  ; #2腔体测试中
; rung 26
@LD W35.11  ; #2腔体破真空结束
OR W35.12  ; #2腔体吹气阀打开
ANDNOT T0019  ; #2合模气缸缩回位延时
OUT W35.12  ; #2腔体吹气阀打开
; rung 27
LD W35.11  ; #2腔体破真空结束
@OR H34.01  ; #2腔体#1位有电池
ANDNOT 9.14  ; #2抽气阀
AND T0389  ; #2腔体破真空值到达
OR W35.13  ; #2合模气缸缩回
ANDNOT W35.00  ; 合模气缸2伸出条件
OUT W35.13  ; #2合模气缸缩回
; rung 28: #2腔体测试结果显示
LD W35.06  ; #2氦检正常结束
OUT TR0
ANDNOT H34.02  ; #2腔体产品NG
@MOV(021) &1 D3208  ; #2腔体测试结果
LD TR0
AND H34.02  ; #2腔体产品NG
@MOV(021) &2 D3208  ; #2腔体测试结果
; rung 29
LD W35.07  ; #2抽气异常结束
@MOV(021) &3 D3208  ; #2腔体测试结果

### Section 真空计及漏率标准转化

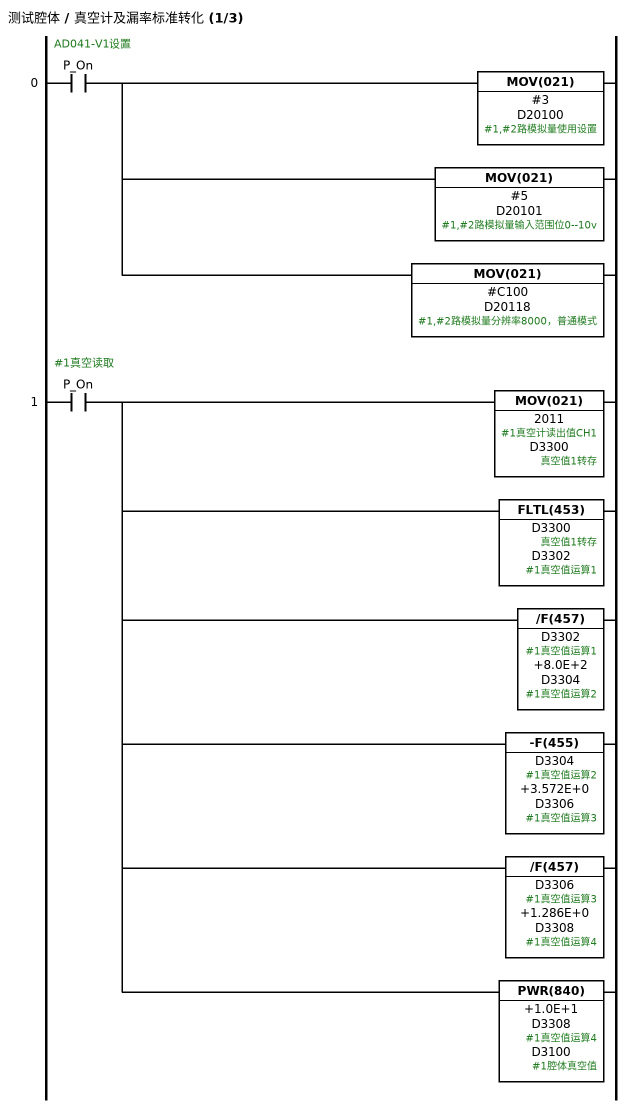
; rung 0: AD041-V1设置
LD P_On
MOV(021) #3 D20100  ; #1,#2路模拟量使用设置
MOV(021) #5 D20101  ; #1,#2路模拟量输入范围位0--10v
MOV(021) #C100 D20118  ; #1,#2路模拟量分辨率8000，普通模式
; rung 1: #1真空读取
LD P_On
MOV(021) 2011 D3300  ; #1真空计读出值CH1, 真空值1转存
FLTL(453) D3300 D3302  ; 真空值1转存, #1真空值运算1
/F(457) D3302 +8.0E+2 D3304  ; #1真空值运算1, #1真空值运算2
-F(455) D3304 +3.572E+0 D3306  ; #1真空值运算2, #1真空值运算3
/F(457) D3306 +1.286E+0 D3308  ; #1真空值运算3, #1真空值运算4
PWR(840) +1.0E+1 D3308 D3100  ; #1真空值运算4, #1腔体真空值

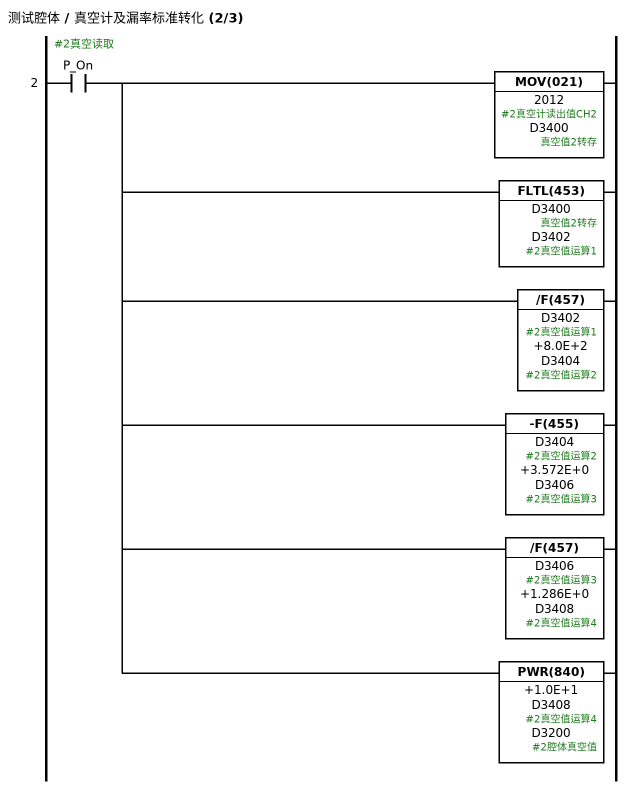
; rung 2: #2真空读取
LD P_On
MOV(021) 2012 D3400  ; #2真空计读出值CH2, 真空值2转存
FLTL(453) D3400 D3402  ; 真空值2转存, #2真空值运算1
/F(457) D3402 +8.0E+2 D3404  ; #2真空值运算1, #2真空值运算2
-F(455) D3404 +3.572E+0 D3406  ; #2真空值运算2, #2真空值运算3
/F(457) D3406 +1.286E+0 D3408  ; #2真空值运算3, #2真空值运算4
PWR(840) +1.0E+1 D3408 D3200  ; #2真空值运算4, #2腔体真空值

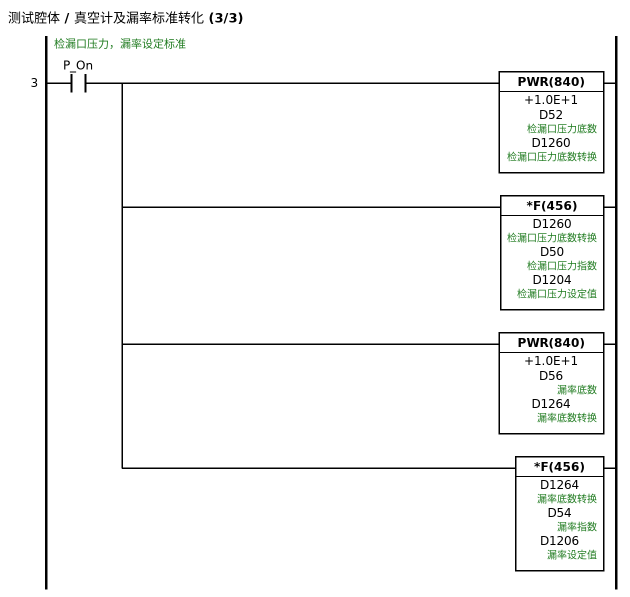
; rung 3: 检漏口压力，漏率设定标准
LD P_On
PWR(840) +1.0E+1 D52 D1260  ; 检漏口压力底数, 检漏口压力底数转换
*F(456) D1260 D50 D1204  ; 检漏口压力底数转换, 检漏口压力指数, 检漏口压力设定值
PWR(840) +1.0E+1 D56 D1264  ; 漏率底数, 漏率底数转换
*F(456) D1264 D54 D1206  ; 漏率底数转换, 漏率指数, 漏率设定值

### Section 氦检仪读值

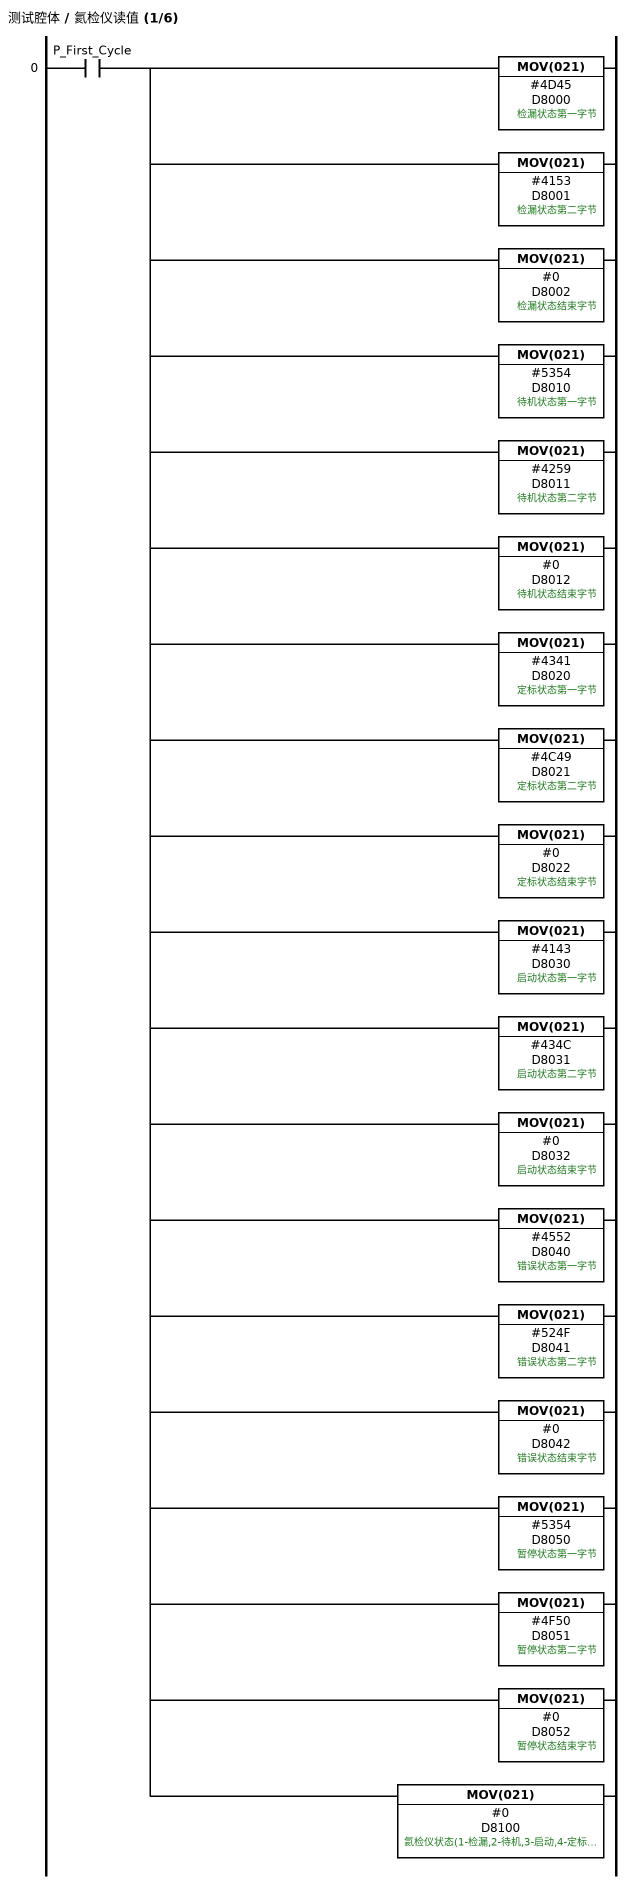
; rung 0
LD P_First_Cycle
MOV(021) #4D45 D8000  ; 检漏状态第一字节
MOV(021) #4153 D8001  ; 检漏状态第二字节
MOV(021) #0 D8002  ; 检漏状态结束字节
MOV(021) #5354 D8010  ; 待机状态第一字节
MOV(021) #4259 D8011  ; 待机状态第二字节
MOV(021) #0 D8012  ; 待机状态结束字节
MOV(021) #4341 D8020  ; 定标状态第一字节
MOV(021) #4C49 D8021  ; 定标状态第二字节
MOV(021) #0 D8022  ; 定标状态结束字节
MOV(021) #4143 D8030  ; 启动状态第一字节
MOV(021) #434C D8031  ; 启动状态第二字节
MOV(021) #0 D8032  ; 启动状态结束字节
MOV(021) #4552 D8040  ; 错误状态第一字节
MOV(021) #524F D8041  ; 错误状态第二字节
MOV(021) #0 D8042  ; 错误状态结束字节
MOV(021) #5354 D8050  ; 暂停状态第一字节
MOV(021) #4F50 D8051  ; 暂停状态第二字节
MOV(021) #0 D8052  ; 暂停状态结束字节
MOV(021) #0 D8100  ; 氦检仪状态(1-检漏,2-待机,3-启动,4-定标,5-错误,6-暂停)

